{attribute 'enable_dynamic_creation'}
// Deferred messages used in case if logging occured when code called using RPC (from ADS client or OPC-UA client, for example) 
FUNCTION_BLOCK INTERNAL DeferredLoggingRecord EXTENDS TwinCAT_OpenFramework_Core.Object
VAR_INPUT
	Level : LOGGING_LEVEL;
	Message : ERROR_MESSAGE;
END_VAR
VAR
	_ClassName : STRING := __POUNAME();
END_VAR

{attribute 'monitoring' := 'call'}
PROPERTY ClassName : STRING
GET
ClassName := _ClassName;
END_GET
END_PROPERTY

{attribute 'monitoring' := 'call'}
PROPERTY Size : ULINT
GET
Size := XSIZEOF(THIS^);
END_GET
END_PROPERTY

END_FUNCTION_BLOCK

(* stored: Version 1.1.0.1
   POU DeferredLoggingRecord: Id {8d29f614-c40c-4f66-b330-979871d888da}, SpecialFunc None
   Property ClassName: Id {b7c162ff-9308-4c0a-839f-24af9cbfe373}
   Get Get: Id {dc14a107-645f-4505-8ac7-0b79164f18f5}
   Property Size: Id {92f45a76-66ab-4026-93d9-0c094dbad523}
   Get Get: Id {d1242558-3b95-48a1-8c7d-04a5dca8537d} *)
